(*
SPDX-FileCopyrightText: © 2026 Oleksandr Tiutyk <trofimich@gmail.com>
SPDX-License-Identifier: MIT
License: https://opensource.org/license/mit
*)

INTERFACE IArgumentTypeClassNotSupportedException EXTENDS IGeneralException

METHOD Throw
VAR_INPUT
	sourceNamespaceName : STRING;
	sourceClassName : STRING;
	sourcePOUName : STRING;
	sourcePosition : STRING;
	argumentName : STRING;
	argumentType : __SYSTEM.TYPE_CLASS;
END_VAR
END_METHOD

END_INTERFACE

(* stored: Version 1.1.0.1
   Itf IArgumentTypeClassNotSupportedException: Id {995b7d02-5c02-41d1-93c2-25c419249058}
   Method Throw: Id {4b5f8966-8659-43ba-a019-abbb92c65cca} *)
